TYPE typeMessageRowsArry :
STRUCT
	
	AlarmViewMsg : ARRAY[1..HMIData.gNumberOfMessagesScreen] OF typeMessageRow;
	WarningViewMsg : ARRAY[1..HMIData.gNumberOfMessagesScreen] OF typeMessageRow;
	PromptViewMsg : ARRAY[1..HMIData.gNumberOfMessagesScreen] OF typeMessageRow;

END_STRUCT
END_TYPE

(* stored: Version 1.1.0.1, ProductVersion 3.1.4024.12
   DUT typeMessageRowsArry: Id {a71a553f-ac0a-4b87-8a43-dbf602736447} *)
